// TIA Portal V18 export
TYPE "TM_Pulse_2x24_Out"
   STRUCT
      Ch0 : "TM_Pulse_2x24_Out_PWM";
      Ch1 { S7_SetPoint := 'True'} : "TM_Pulse_2x24_Out_PWM";
   END_STRUCT;
END_TYPE
